Xinje XDPPro project, PLC1: XD3-16 (software 3.7.17b 2023-10-13)

PROGRAM Ladder

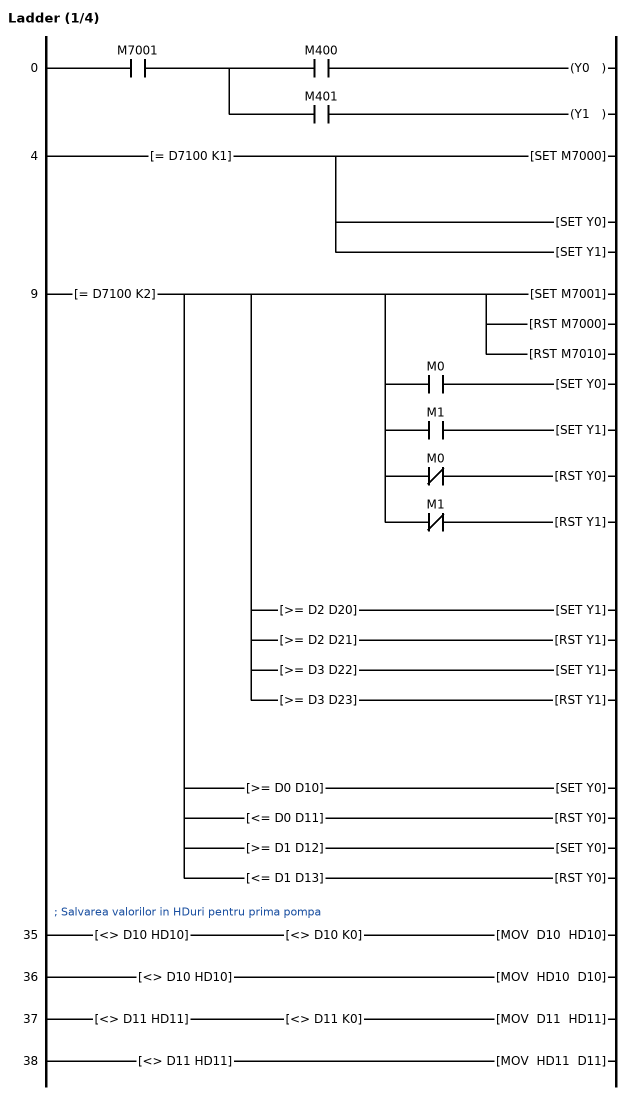
LD     M7001
MPS
AND    M400
OUT    Y0
MPP
AND    M401
OUT    Y1
LD=    D7100 K1
SET    M7000
SET    Y0
SET    Y1
LD=    D7100 K2
SET    M7001
RST    M7000
RST    M7010
MPS
AND    M0
SET    Y0
MRD
AND    M1
SET    Y1
MRD
ANI    M0
RST    Y0
MRD
ANI    M1
RST    Y1
MRD
AND>=  D2 D20
SET    Y1
MRD
AND>=  D2 D21
RST    Y1
MRD
AND>=  D3 D22
SET    Y1
MRD
AND>=  D3 D23
RST    Y1
MRD
AND>=  D0 D10
SET    Y0
MRD
AND<=  D0 D11
RST    Y0
MRD
AND>=  D1 D12
SET    Y0
MPP
AND<=  D1 D13
RST    Y0
; Salvarea valorilor in HDuri pentru prima pompa
LD<>   D10 HD10
AND<>  D10 K0
MOV    D10 HD10
LD<>   D10 HD10
MOV    HD10 D10
LD<>   D11 HD11
AND<>  D11 K0
MOV    D11 HD11
LD<>   D11 HD11
MOV    HD11 D11

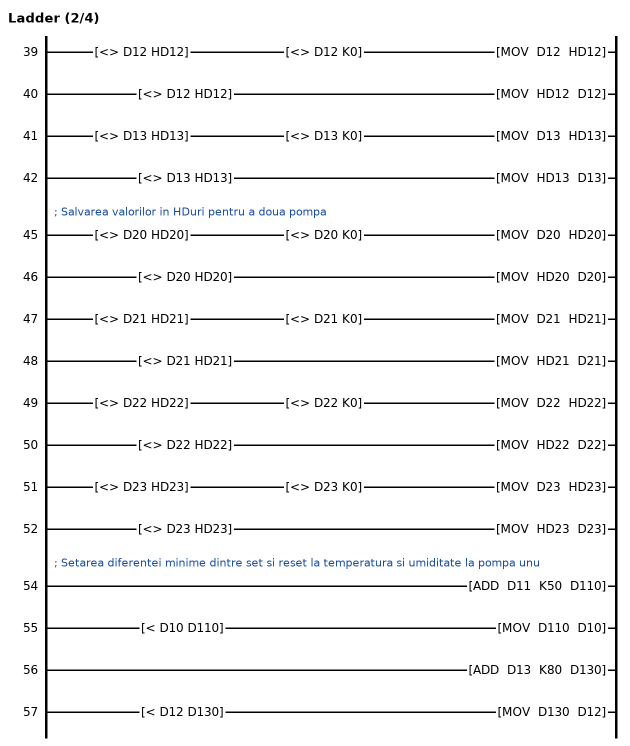
LD<>   D12 HD12
AND<>  D12 K0
MOV    D12 HD12
LD<>   D12 HD12
MOV    HD12 D12
LD<>   D13 HD13
AND<>  D13 K0
MOV    D13 HD13
LD<>   D13 HD13
MOV    HD13 D13
; Salvarea valorilor in HDuri pentru a doua pompa
LD<>   D20 HD20
AND<>  D20 K0
MOV    D20 HD20
LD<>   D20 HD20
MOV    HD20 D20
LD<>   D21 HD21
AND<>  D21 K0
MOV    D21 HD21
LD<>   D21 HD21
MOV    HD21 D21
LD<>   D22 HD22
AND<>  D22 K0
MOV    D22 HD22
LD<>   D22 HD22
MOV    HD22 D22
LD<>   D23 HD23
AND<>  D23 K0
MOV    D23 HD23
LD<>   D23 HD23
MOV    HD23 D23
; Setarea diferentei minime dintre set si reset la temperatura si umiditate la pompa unu
ADD    D11 K50 D110
LD<    D10 D110
MOV    D110 D10
ADD    D13 K80 D130
LD<    D12 D130
MOV    D130 D12

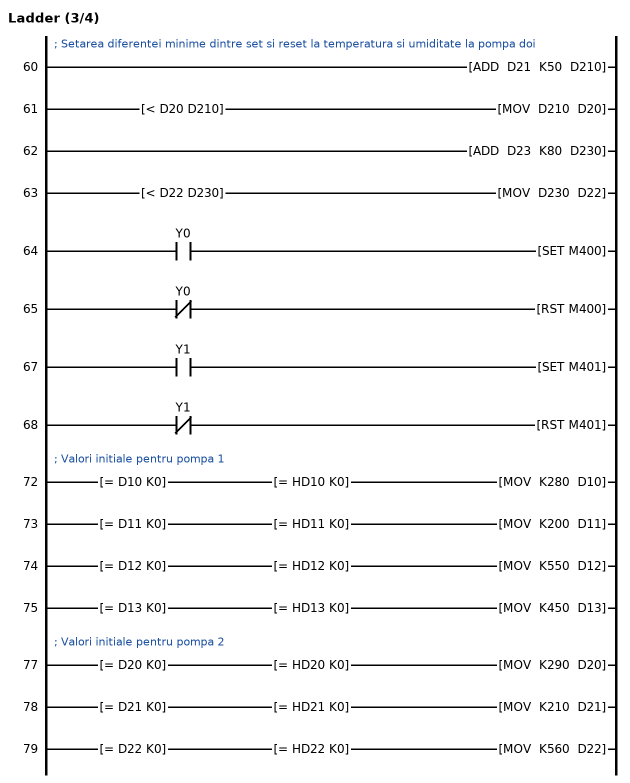
; Setarea diferentei minime dintre set si reset la temperatura si umiditate la pompa doi
ADD    D21 K50 D210
LD<    D20 D210
MOV    D210 D20
ADD    D23 K80 D230
LD<    D22 D230
MOV    D230 D22
LD     Y0
SET    M400
LDI    Y0
RST    M400
LD     Y1
SET    M401
LDI    Y1
RST    M401
; Valori initiale pentru pompa 1
LD=    D10 K0
AND=   HD10 K0
MOV    K280 D10
LD=    D11 K0
AND=   HD11 K0
MOV    K200 D11
LD=    D12 K0
AND=   HD12 K0
MOV    K550 D12
LD=    D13 K0
AND=   HD13 K0
MOV    K450 D13
; Valori initiale pentru pompa 2
LD=    D20 K0
AND=   HD20 K0
MOV    K290 D20
LD=    D21 K0
AND=   HD21 K0
MOV    K210 D21
LD=    D22 K0
AND=   HD22 K0
MOV    K560 D22

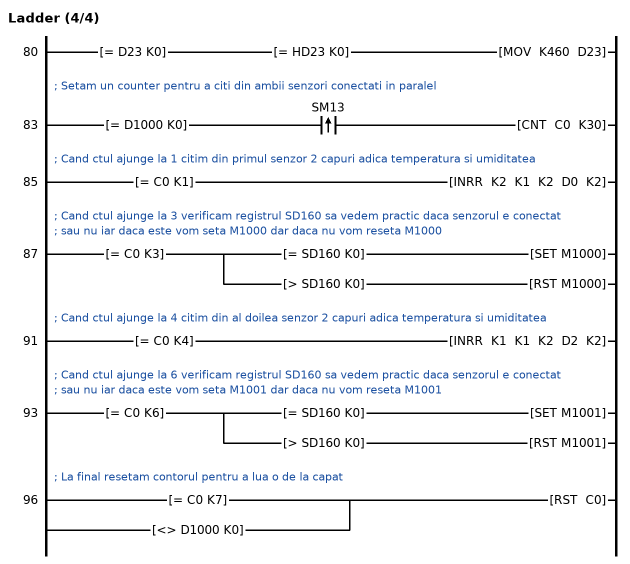
LD=    D23 K0
AND=   HD23 K0
MOV    K460 D23
; Setam un counter pentru a citi din ambii senzori conectati in paralel
LD=    D1000 K0
ANDP   SM13
CNT    C0 K30
; Cand ctul ajunge la 1 citim din primul senzor 2 capuri adica temperatura si umiditatea
LD=    C0 K1
INRR   K2 K1 K2 D0 K2
; Cand ctul ajunge la 3 verificam registrul SD160 sa vedem practic daca senzorul e conectat sau nu iar daca este vom seta M1000 dar daca nu vom reseta M1000
LD=    C0 K3
MPS
AND=   SD160 K0
SET    M1000
MPP
AND>   SD160 K0
RST    M1000
; Cand ctul ajunge la 4 citim din al doilea senzor 2 capuri adica temperatura si umiditatea
LD=    C0 K4
INRR   K1 K1 K2 D2 K2
; Cand ctul ajunge la 6 verificam registrul SD160 sa vedem practic daca senzorul e conectat sau nu iar daca este vom seta M1001 dar daca nu vom reseta M1001
LD=    C0 K6
MPS
AND=   SD160 K0
SET    M1001
MPP
AND>   SD160 K0
RST    M1001
; La final resetam contorul pentru a lua o de la capat
LD=    C0 K7
OR<>   D1000 K0
RST    C0